{attribute 'GeneratedUsingTerminal: IODEVICETYPE_ETHERCATPROT'}
{attribute addProperty BoxType "IODEVICETYPE_ETHERCATPROT"}
{attribute addProperty Id "Beckhoff_EJ1xxxBeckhoff_EJ1xxx_8ABA4DFB121Beckhoff_EJ2xxxBeckhoff_EJ2xxx_F745D3BC254Beckhoff_EJ3xxxBeckhoff_EJ3xxx_FBC884521180Beckhoff_EJ4xxxBeckhoff_EJ4xxx_A145C67B177Beckhoff_EJ5xxxBeckhoff_EJ5xxx_E1A62FB7142Beckhoff_EJ6xxxBeckhoff_EJ6xxx_D380D5DE176Beckhoff_EJ7xxxBeckhoff_EJ7xxx_D0F87F471315Beckhoff_EJ9xxxBeckhoff_EJ9xxx_491FB8F7124Beckhoff_EJx9xxBeckhoff_EJx9xx_66D9432D462SyncUnitsSyncUnits_99E584AF18InputsInputs_25A0042B160OutputsOutputs_2397A10E106InfoDataInfoData_E68C61CD28"}
{attribute addProperty CRC "1846226854"}
{attribute addProperty Size "4263"}
TYPE EtherCAT_Master_EJxxxx_6E0B2FA6 :
STRUCT
	{attribute addProperty Name "Beckhoff_EJ1xxx"}
	{attribute addProperty PreviousPort "EtherCAT_Master_EJxxxx : Master"}
	Beckhoff_EJ1xxx : Beckhoff_EJ1xxx_8ABA4DFB;
	{attribute addProperty Name "Beckhoff_EJ2xxx"}
	{attribute addProperty PreviousPort "Beckhoff EJ1xxx : C"}
	Beckhoff_EJ2xxx : Beckhoff_EJ2xxx_F745D3BC;
	{attribute addProperty Name "Beckhoff_EJ3xxx"}
	{attribute addProperty PreviousPort "Beckhoff EJ2xxx : C"}
	Beckhoff_EJ3xxx : Beckhoff_EJ3xxx_FBC88452;
	{attribute addProperty Name "Beckhoff_EJ4xxx"}
	{attribute addProperty PreviousPort "Beckhoff EJ3xxx : C"}
	Beckhoff_EJ4xxx : Beckhoff_EJ4xxx_A145C67B;
	{attribute addProperty Name "Beckhoff_EJ5xxx"}
	{attribute addProperty PreviousPort "Beckhoff EJ4xxx : C"}
	Beckhoff_EJ5xxx : Beckhoff_EJ5xxx_E1A62FB7;
	{attribute addProperty Name "Beckhoff_EJ6xxx"}
	{attribute addProperty PreviousPort "Beckhoff EJ5xxx : C"}
	Beckhoff_EJ6xxx : Beckhoff_EJ6xxx_D380D5DE;
	{attribute addProperty Name "Beckhoff_EJ7xxx"}
	{attribute addProperty PreviousPort "Beckhoff EJ6xxx : C"}
	Beckhoff_EJ7xxx : Beckhoff_EJ7xxx_D0F87F47;
	{attribute addProperty Name "Beckhoff_EJ9xxx"}
	{attribute addProperty PreviousPort "Beckhoff EJ7xxx : C"}
	Beckhoff_EJ9xxx : Beckhoff_EJ9xxx_491FB8F7;
	{attribute addProperty Name "Beckhoff_EJx9xx"}
	{attribute addProperty PreviousPort "Beckhoff EJ9xxx : C"}
	Beckhoff_EJx9xx : Beckhoff_EJx9xx_66D9432D;
	{attribute addProperty Name "SyncUnits"}
	SyncUnits : SyncUnits_99E584AF;
	{attribute addProperty Name "Inputs"}
	Inputs : Inputs_25A0042B;
	{attribute addProperty Name "Outputs"}
	Outputs : Outputs_2397A10E;
	{attribute addProperty Name "InfoData"}
	InfoData : InfoData_E68C61CD;
END_STRUCT
END_TYPE

(* stored: Version 1.2.0.0, ProductVersion 3.1.4024.9
   DUT EtherCAT_Master_EJxxxx_6E0B2FA6: Id {8d3e4d7c-61df-4427-8111-b57c4f0ded8f} *)
